// Bergplaats B1-11L0-00
TYPE ST_WP_StorageRoom :
STRUCT
	fbButton1		: FB_DigitalIn;
	fbButton2		: FB_DigitalIn;
	fbButton3		: FB_DigitalIn;
END_STRUCT
END_TYPE

(* stored: Version 1.1.0.1, ProductVersion 3.1.4024.12
   DUT ST_WP_StorageRoom: Id {e559ad85-825d-4706-9246-b63935192fbf} *)
